TYPE XINPUT_GAMEPAD :
STRUCT
 wButtons: WORD;
 bLeftTrigger: BYTE;
 bRightTrigger: BYTE;
 sThumbLX: INT;
 sThumbLY: INT;
 sThumbRX: INT;
 sThumbRY: INT;
END_STRUCT
END_TYPE

(* stored: Version 1.1.0.1, ProductVersion 3.1.4024.10
   DUT XINPUT_GAMEPAD: Id {d5ddfd97-d709-462c-8a37-f8650f1e26fe} *)
